% RSLogix 500 project I2P JOB 15 ALEXANDER_LOYND_BAK069.RSS, saved by version 10.00.00.00 %
PROJECT "ML06A"    % processor: Bul.1763 MicroLogix 1100 Series B %

PROGRAM FILES
  LAD 2   16 rungs

DATA FILES
  O0 OUTPUT  4 elements
  I1 INPUT  6 elements
  S2 STATUS  66 elements
  B3 BINARY  1 elements
  T4 TIMER  2 elements
  C5 COUNTER  1 elements
  R6 CONTROL  1 elements
  N7 INTEGER  1 elements
  F8 FLOAT  1 elements

LADDER 2
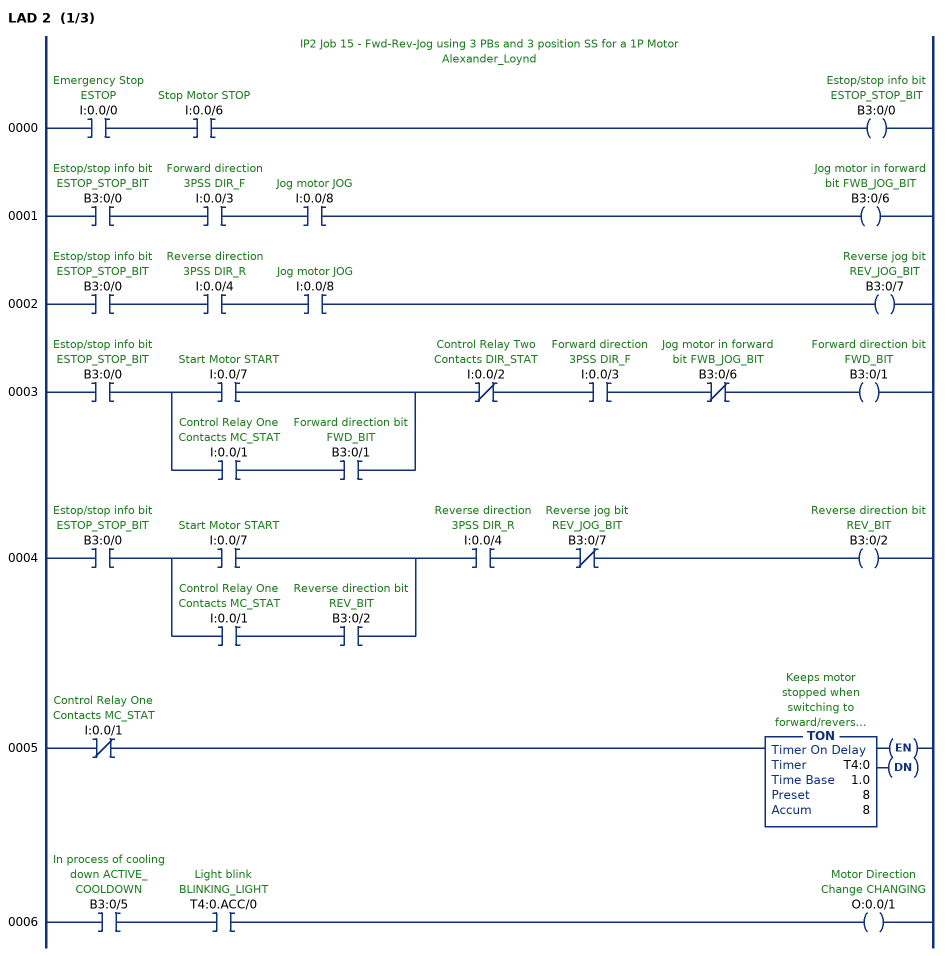
% Rung: 0 %
% IP2 Job 15 - Fwd-Rev-Jog using 3 PBs and 3 position SS for a 1P Motor
% Alexander_Loynd %
SOR XIC I:0.0/0 XIC I:0.0/6 OTE B3:0/0 EOR
%   I:0.0/0  ESTOP  "Emergency Stop" %
%   I:0.0/6  STOP  "Stop Motor" %
%   B3:0/0  ESTOP_STOP_BIT  "Estop/stop info bit" %
% Rung: 1 %
SOR XIC B3:0/0 XIC I:0.0/3 XIC I:0.0/8 OTE B3:0/6 EOR
%   B3:0/0  ESTOP_STOP_BIT  "Estop/stop info bit" %
%   I:0.0/3  DIR_F  "Forward direction 3PSS" %
%   I:0.0/8  JOG  "Jog motor" %
%   B3:0/6  FWB_JOG_BIT  "Jog motor in forward bit" %
% Rung: 2 %
SOR XIC B3:0/0 XIC I:0.0/4 XIC I:0.0/8 OTE B3:0/7 EOR
%   B3:0/0  ESTOP_STOP_BIT  "Estop/stop info bit" %
%   I:0.0/4  DIR_R  "Reverse direction 3PSS" %
%   I:0.0/8  JOG  "Jog motor" %
%   B3:0/7  REV_JOG_BIT  "Reverse jog bit" %
% Rung: 3 %
SOR XIC B3:0/0 BST XIC I:0.0/7 NXB XIC I:0.0/1 XIC B3:0/1 BND XIO I:0.0/2 XIC I:0.0/3 XIO B3:0/6 OTE B3:0/1 EOR
%   B3:0/0  ESTOP_STOP_BIT  "Estop/stop info bit" %
%   I:0.0/7  START  "Start Motor" %
%   I:0.0/1  MC_STAT  "Control Relay One Contacts" %
%   B3:0/1  FWD_BIT  "Forward direction bit" %
%   I:0.0/2  DIR_STAT  "Control Relay Two Contacts" %
%   I:0.0/3  DIR_F  "Forward direction 3PSS" %
%   B3:0/6  FWB_JOG_BIT  "Jog motor in forward bit" %
% Rung: 4 %
SOR XIC B3:0/0 BST XIC I:0.0/7 NXB XIC I:0.0/1 XIC B3:0/2 BND XIC I:0.0/4 XIO B3:0/7 OTE B3:0/2 EOR
%   B3:0/0  ESTOP_STOP_BIT  "Estop/stop info bit" %
%   I:0.0/7  START  "Start Motor" %
%   I:0.0/1  MC_STAT  "Control Relay One Contacts" %
%   B3:0/2  REV_BIT  "Reverse direction bit" %
%   I:0.0/4  DIR_R  "Reverse direction 3PSS" %
%   B3:0/7  REV_JOG_BIT  "Reverse jog bit" %
% Rung: 5 %
SOR XIO I:0.0/1 TON T4:0 1.0 8 8 EOR
%   I:0.0/1  MC_STAT  "Control Relay One Contacts" %
%   T4:0  MTR_DELAY  "Keeps motor stopped when switching to forward/reverse" %
% Rung: 6 %
SOR XIC B3:0/5 XIC T4:0.ACC/0 OTE O:0.0/1 EOR
%   B3:0/5  ACTIVE_COOLDOWN  "In process of cooling down" %
%   T4:0.ACC/0  BLINKING_LIGHT  "Light blink" %
%   O:0.0/1  CHANGING  "Motor Direction Change" %

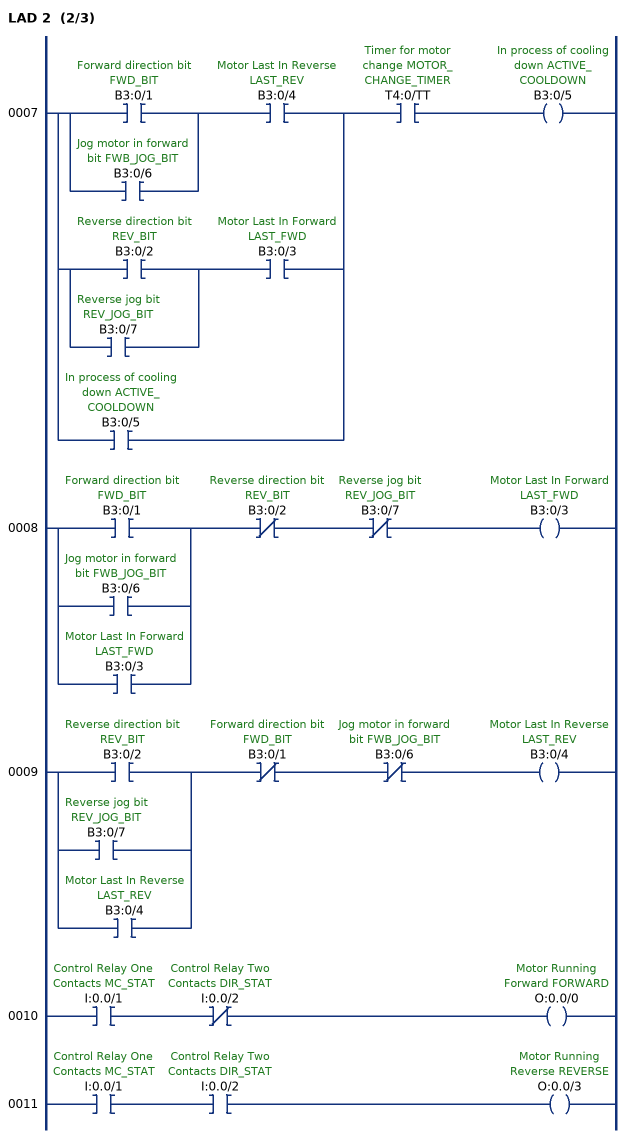
% Rung: 7 %
SOR BST BST XIC B3:0/1 NXB XIC B3:0/6 BND XIC B3:0/4 NXB BST XIC B3:0/2 NXB XIC B3:0/7 BND XIC B3:0/3 NXB XIC B3:0/5 BND XIC T4:0/TT OTE B3:0/5 EOR
%   B3:0/1  FWD_BIT  "Forward direction bit" %
%   B3:0/6  FWB_JOG_BIT  "Jog motor in forward bit" %
%   B3:0/4  LAST_REV  "Motor Last In Reverse" %
%   B3:0/2  REV_BIT  "Reverse direction bit" %
%   B3:0/7  REV_JOG_BIT  "Reverse jog bit" %
%   B3:0/3  LAST_FWD  "Motor Last In Forward" %
%   B3:0/5  ACTIVE_COOLDOWN  "In process of cooling down" %
%   T4:0/TT  MOTOR_CHANGE_TIMER  "Timer for motor change" %
% Rung: 8 %
SOR BST BST XIC B3:0/1 NXB XIC B3:0/6 BND NXB XIC B3:0/3 BND XIO B3:0/2 XIO B3:0/7 OTE B3:0/3 EOR
%   B3:0/1  FWD_BIT  "Forward direction bit" %
%   B3:0/6  FWB_JOG_BIT  "Jog motor in forward bit" %
%   B3:0/3  LAST_FWD  "Motor Last In Forward" %
%   B3:0/2  REV_BIT  "Reverse direction bit" %
%   B3:0/7  REV_JOG_BIT  "Reverse jog bit" %
% Rung: 9 %
SOR BST BST XIC B3:0/2 NXB XIC B3:0/7 BND NXB XIC B3:0/4 BND XIO B3:0/1 XIO B3:0/6 OTE B3:0/4 EOR
%   B3:0/2  REV_BIT  "Reverse direction bit" %
%   B3:0/7  REV_JOG_BIT  "Reverse jog bit" %
%   B3:0/4  LAST_REV  "Motor Last In Reverse" %
%   B3:0/1  FWD_BIT  "Forward direction bit" %
%   B3:0/6  FWB_JOG_BIT  "Jog motor in forward bit" %
% Rung: 10 %
SOR XIC I:0.0/1 XIO I:0.0/2 OTE O:0.0/0 EOR
%   I:0.0/1  MC_STAT  "Control Relay One Contacts" %
%   I:0.0/2  DIR_STAT  "Control Relay Two Contacts" %
%   O:0.0/0  FORWARD  "Motor Running Forward" %
% Rung: 11 %
SOR XIC I:0.0/1 XIC I:0.0/2 OTE O:0.0/3 EOR
%   I:0.0/1  MC_STAT  "Control Relay One Contacts" %
%   I:0.0/2  DIR_STAT  "Control Relay Two Contacts" %
%   O:0.0/3  REVERSE  "Motor Running Reverse" %

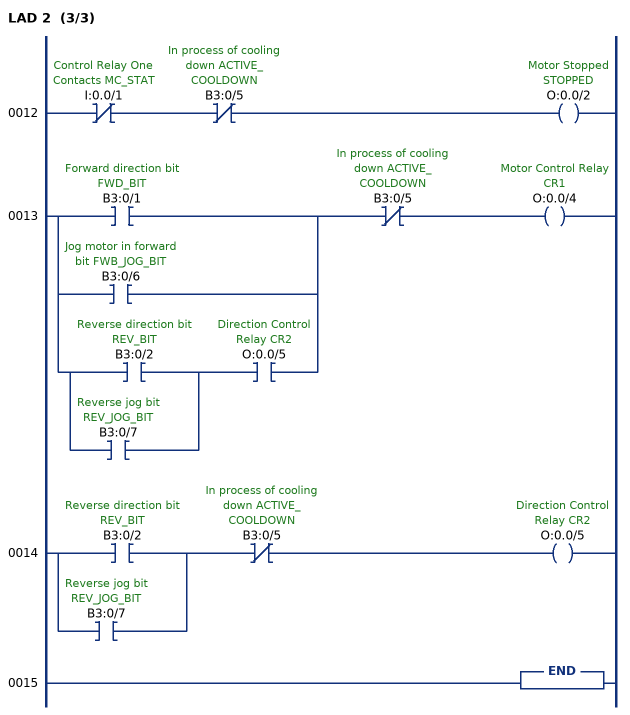
% Rung: 12 %
SOR XIO I:0.0/1 XIO B3:0/5 OTE O:0.0/2 EOR
%   I:0.0/1  MC_STAT  "Control Relay One Contacts" %
%   B3:0/5  ACTIVE_COOLDOWN  "In process of cooling down" %
%   O:0.0/2  STOPPED  "Motor Stopped" %
% Rung: 13 %
SOR BST BST XIC B3:0/1 NXB XIC B3:0/6 BND NXB BST XIC B3:0/2 NXB XIC B3:0/7 BND XIC O:0.0/5 BND XIO B3:0/5 OTE O:0.0/4 EOR
%   B3:0/1  FWD_BIT  "Forward direction bit" %
%   B3:0/6  FWB_JOG_BIT  "Jog motor in forward bit" %
%   B3:0/2  REV_BIT  "Reverse direction bit" %
%   B3:0/7  REV_JOG_BIT  "Reverse jog bit" %
%   O:0.0/5  CR2  "Direction Control Relay" %
%   B3:0/5  ACTIVE_COOLDOWN  "In process of cooling down" %
%   O:0.0/4  CR1  "Motor Control Relay" %
% Rung: 14 %
SOR BST XIC B3:0/2 NXB XIC B3:0/7 BND XIO B3:0/5 OTE O:0.0/5 EOR
%   B3:0/2  REV_BIT  "Reverse direction bit" %
%   B3:0/7  REV_JOG_BIT  "Reverse jog bit" %
%   B3:0/5  ACTIVE_COOLDOWN  "In process of cooling down" %
%   O:0.0/5  CR2  "Direction Control Relay" %
% Rung: 15 %
SOR END EOR

OTHER DOCUMENTED ADDRESSES
  I:0.0/5  RUN_JOG  "Run/Jog Mode"
  PB1  "Start Motor"
  T4:1/DN  TIMER_DONE  "timer hit done"
  T4:1/TT  TIMER_TIMING  "Timer timeing"

DATA TABLE (non-zero values as saved)
DATA B3
% B3:0 % 0X0011
DATA T4
% .PRE .ACC %
% T4:0 % 8 8
% T4:1 % 1 0
